// Mitsubishi GX Works2 project: IELET2103_Datalab6   PLC: FX2N/FX2NC
// IELET2103_Datalab6

// global labels: Global1
VAR_GLOBAL
  Stopp AT X000 : BOOL;
  Start AT X001 : BOOL;
  EndestillingA AT X002 : BOOL;
  MidtstillingB AT X003 : BOOL;
  EndestillingC AT X004 : BOOL;
  VognFrem AT Y000 : BOOL;
  VognTilbake AT Y001 : BOOL;
  EndestillingStengtSpjeld AT X005 : BOOL;
  EndestillingAapentSpjeld AT X006 : BOOL;
  MagnetventilForAapningAvSpjeld AT Y002 : BOOL;
  MagnetventilForLukkingAvSpjeld AT Y003 : BOOL;
END_VAR

// task Task_01 (event TRUE, interval 0, priority 31): Oppgave1c)

PROGRAM Oppgave1a)
(* structured ladder/FBD written out as ST: instructions are called as NAME(EN, inputs, outputs); _pN, _eN, _tN stand for wires *)
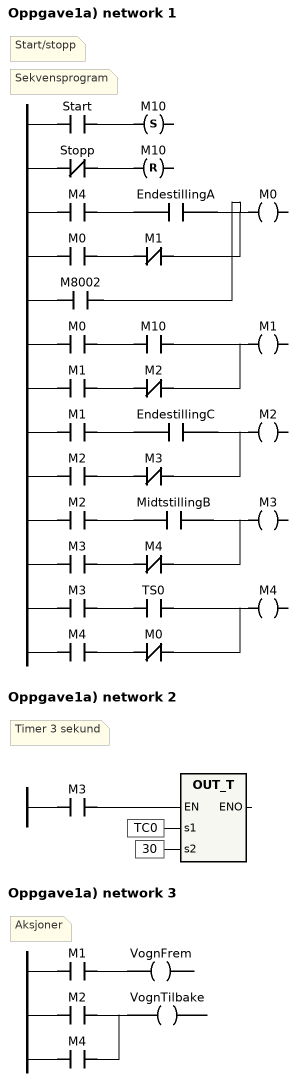
(* network 1 *)
(* Start/stopp *)
(* Sekvensprogram *)
SET(Start, M10);
RST(NOT Stopp, M10);
M0 := (M4 AND EndestillingA) OR (M0 AND NOT M1) OR M8002;
M1 := (M0 AND M10) OR (M1 AND NOT M2);
M2 := (M1 AND EndestillingC) OR (M2 AND NOT M3);
M3 := (M2 AND MidtstillingB) OR (M3 AND NOT M4);
M4 := (M3 AND TS0) OR (M4 AND NOT M0);
(* network 2 *)
(* Timer 3 sekund *)
OUT_T(M3, TC0, 30);
(* network 3 *)
(* Aksjoner *)
VognFrem := M1;
VognTilbake := M2 OR M4;
END_PROGRAM

PROGRAM Oppgave1c)
(* structured ladder/FBD written out as ST: instructions are called as NAME(EN, inputs, outputs); _pN, _eN, _tN stand for wires *)
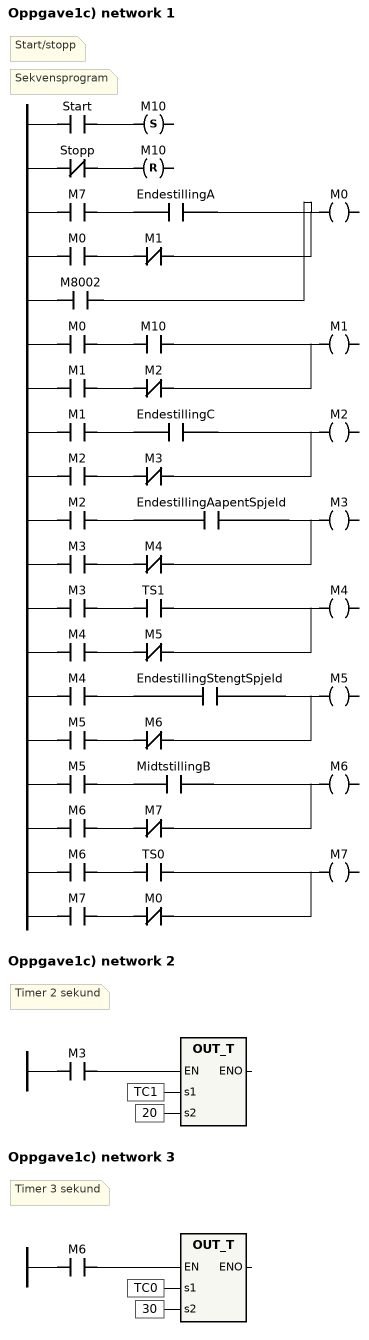
(* network 1 *)
(* Start/stopp *)
(* Sekvensprogram *)
SET(Start, M10);
RST(NOT Stopp, M10);
M0 := (M7 AND EndestillingA) OR (M0 AND NOT M1) OR M8002;
M1 := (M0 AND M10) OR (M1 AND NOT M2);
M2 := (M1 AND EndestillingC) OR (M2 AND NOT M3);
M3 := (M2 AND EndestillingAapentSpjeld) OR (M3 AND NOT M4);
M4 := (M3 AND TS1) OR (M4 AND NOT M5);
M5 := (M4 AND EndestillingStengtSpjeld) OR (M5 AND NOT M6);
M6 := (M5 AND MidtstillingB) OR (M6 AND NOT M7);
M7 := (M6 AND TS0) OR (M7 AND NOT M0);
(* network 2 *)
(* Timer 2 sekund *)
OUT_T(M3, TC1, 20);
(* network 3 *)
(* Timer 3 sekund *)
OUT_T(M6, TC0, 30);
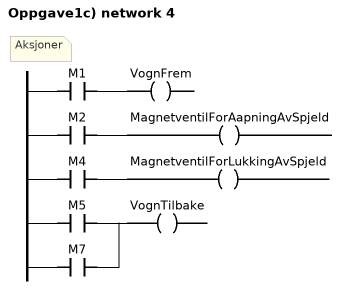
(* network 4 *)
(* Aksjoner *)
VognFrem := M1;
MagnetventilForAapningAvSpjeld := M2;
MagnetventilForLukkingAvSpjeld := M4;
VognTilbake := M5 OR M7;
END_PROGRAM
